FUNCTION_BLOCK FB_DriveInterface
VAR_INPUT
END_VAR
VAR_OUTPUT
END_VAR
VAR
	power: MC_Power; //MC_Power instance
	reset: MC_Reset;
	moveabs: MC_MoveAbsolute;
	moverel: MC_MoveRelative;
	stop: MC_Stop;
	setOverride: MC_SetOverride;
END_VAR

VAR_IN_OUT
	plcAxis:typeDriveInterface; //axis ref to the rest of PLC
	ncAxis:axis_ref; //axis ref of the NC drive (only beckhoff)
	
END_VAR

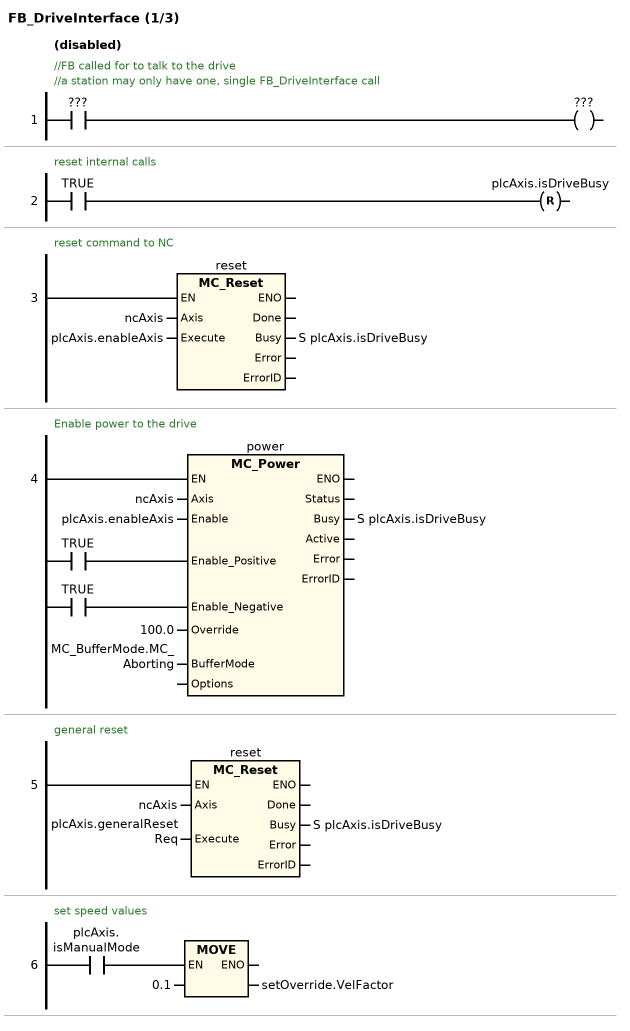
// NETWORK 1 (disabled)
// //FB called for to talk to the drive
// //a station may only have one, single FB_DriveInterface call
// ??? := ???;

// NETWORK 2
// reset internal calls
plcAxis.isDriveBusy R= TRUE;

// NETWORK 3
// reset command to NC
reset(Axis := ncAxis, Execute := plcAxis.enableAxis); // MC_Reset
plcAxis.isDriveBusy S= reset.Busy;

// NETWORK 4
// Enable power to the drive
power(
    Axis := ncAxis,
    Enable := plcAxis.enableAxis,
    Enable_Positive := TRUE,
    Enable_Negative := TRUE,
    Override := 100.0,
    BufferMode := MC_BufferMode.MC_Aborting); // MC_Power
plcAxis.isDriveBusy S= power.Busy;

// NETWORK 5
// general reset
reset(Axis := ncAxis, Execute := plcAxis.generalResetReq); // MC_Reset
plcAxis.isDriveBusy S= reset.Busy;

// NETWORK 6
// set speed values
IF plcAxis.isManualMode THEN setOverride.VelFactor := 0.1; END_IF

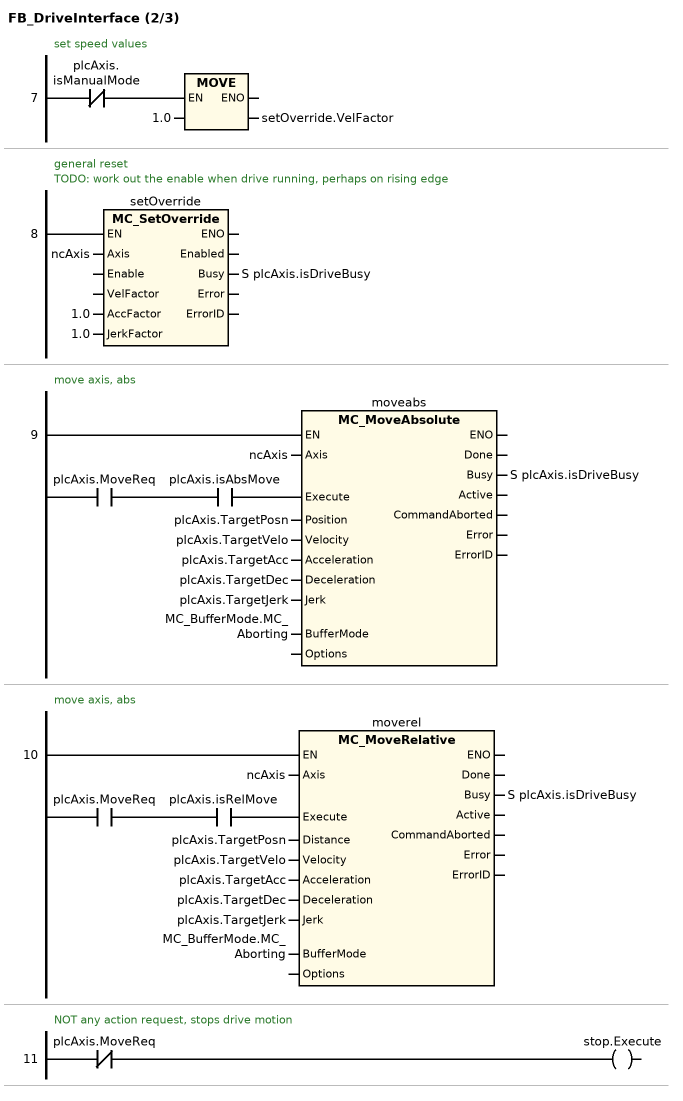
// NETWORK 7
// set speed values
IF NOT plcAxis.isManualMode THEN setOverride.VelFactor := 1.0; END_IF

// NETWORK 8
// general reset
// TODO: work out the enable when drive running, perhaps on rising edge
setOverride(Axis := ncAxis, AccFactor := 1.0, JerkFactor := 1.0); // MC_SetOverride
plcAxis.isDriveBusy S= setOverride.Busy;

// NETWORK 9
// move axis, abs
moveabs(
    Axis := ncAxis,
    Execute := plcAxis.MoveReq AND plcAxis.isAbsMove,
    Position := plcAxis.TargetPosn,
    Velocity := plcAxis.TargetVelo,
    Acceleration := plcAxis.TargetAcc,
    Deceleration := plcAxis.TargetDec,
    Jerk := plcAxis.TargetJerk,
    BufferMode := MC_BufferMode.MC_Aborting); // MC_MoveAbsolute
plcAxis.isDriveBusy S= moveabs.Busy;

// NETWORK 10
//  move axis, abs
moverel(
    Axis := ncAxis,
    Execute := plcAxis.MoveReq AND plcAxis.isRelMove,
    Distance := plcAxis.TargetPosn,
    Velocity := plcAxis.TargetVelo,
    Acceleration := plcAxis.TargetAcc,
    Deceleration := plcAxis.TargetDec,
    Jerk := plcAxis.TargetJerk,
    BufferMode := MC_BufferMode.MC_Aborting); // MC_MoveRelative
plcAxis.isDriveBusy S= moverel.Busy;

// NETWORK 11
// NOT any action request, stops drive motion
stop.Execute := NOT plcAxis.MoveReq;

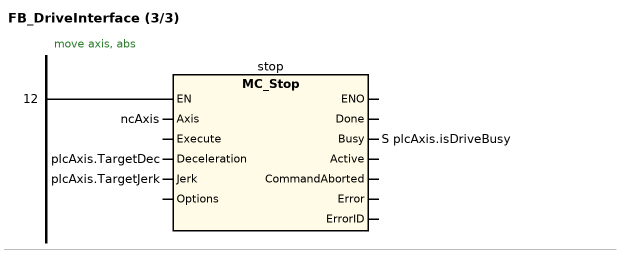
// NETWORK 12
// move axis, abs
stop(Axis := ncAxis, Deceleration := plcAxis.TargetDec, Jerk := plcAxis.TargetJerk); // MC_Stop
plcAxis.isDriveBusy S= stop.Busy;

END_FUNCTION_BLOCK

(* stored: Version 1.1.0.1, ProductVersion 3.1.4024.12
   POU FB_DriveInterface: Id {ef5a2760-99ed-4752-b6d0-8e47bd4f419b}, SpecialFunc None *)
